{attribute 'qualified_only' := ''}
{attribute 'strict' := ''}
TYPE MC_ExecutionMode :
(
	mcImmediatly := 0,
	mcQueue := 1
);
END_TYPE

(* stored: Version 1.1.0.1, ProductVersion 3.1.4024.11
   DUT MC_ExecutionMode: Id {1a4da23f-a449-494b-9033-d06fa4cc943a} *)
